FUNCTION_BLOCK GearTask IMPLEMENTS I_Task, I_Object, I_Abortable, I_Cyclic
VAR
	mcGearIn : MC_GearIn;
	mcGearOut : MC_GearOut;
	_AxisMaster : REFERENCE TO Tc2_MC2.AXIS_REF;
	_Axis : REFERENCE TO Tc2_MC2.AXIS_REF;
END_VAR

METHOD Abort : Base_Library.HRESULT
mcGearIn.Execute := FALSE;
mcGearOut.Execute := FALSE;
END_METHOD

PROPERTY PUBLIC Acceleration : mc_lreal
GET
Acceleration := mcGearIn.Acceleration;
END_GET
SET
mcGearIn.Acceleration := Acceleration;
END_SET
END_PROPERTY

PROPERTY Busy : BOOL
GET
Busy := mcGearIn.Busy OR mcGearOut.Busy;
END_GET
END_PROPERTY

METHOD Cycle : Base_Library.HRESULT
mcGearIn(Master := _AxisMaster, Slave := _Axis);
mcGearOut(Slave := _Axis);
END_METHOD

PROPERTY PUBLIC Deceleration : mc_lreal
GET
Deceleration := mcGearIn.Deceleration;
END_GET
SET
mcGearIn.Deceleration := Deceleration;
END_SET
END_PROPERTY

PROPERTY Done : BOOL
GET
Done := not mcGearIn.Busy OR NOT mcGearOut.Busy;
END_GET
END_PROPERTY

PROPERTY Error : BOOL
GET
Error := mcGearIn.Error OR mcGearOut.Error;
END_GET
END_PROPERTY

METHOD GearIn : BOOL
VAR_INPUT
END_VAR
IF _Axis.Status.NotMoving AND NOT _Axis.Status.Coupled THEN
	mcGearIn.Execute := TRUE;
END_IF
END_METHOD

METHOD GearOut : BOOL
VAR_INPUT
END_VAR
IF _Axis.Status.NotMoving AND _Axis.Status.Coupled THEN
	mcGearOut.Execute := TRUE;
END_IF
END_METHOD

PROPERTY InGear : BOOL
GET
END_GET
END_PROPERTY

PROPERTY PUBLIC Jerk : mc_lreal
GET
Jerk := mcGearIn.Jerk;
END_GET
SET
mcGearIn.Jerk := Jerk;
END_SET
END_PROPERTY

METHOD RegisterWithParent
VAR_INPUT
	Runner	: Base_Library.I_HostObjects;
END_VAR
Runner.RegisterAbortable(THIS^);
Runner.RegisterCyclic(THIS^);
Runner.RegisterTask(This^);
END_METHOD

END_FUNCTION_BLOCK

(* stored: Version 1.1.0.1
   POU GearTask: Id {c68427ee-fbb2-4955-87f7-236eb5ca7453}, SpecialFunc None
   Method Abort: Id {b070cc04-b789-4192-a434-c23424a575ce}
   Property Acceleration: Id {f01bc33a-2696-4e8f-90b9-30cdb8f4dd2d}
   Get Get: Id {b978d70b-e2e1-4621-bbee-98b107797754}
   Set Set: Id {bf531977-c15d-49ee-be06-c4bf1afca554}
   Property Busy: Id {ebe05db7-1dd0-4727-938c-463df03890a3}
   Get Get: Id {c269a663-4580-4d6d-be8e-3ee03a475cea}
   Method Cycle: Id {f8090c6e-65b8-4fad-b206-c4a3dca766fd}
   Property Deceleration: Id {92ba61af-a15e-46bf-86f4-eb6ef3fa3283}
   Get Get: Id {45a7a481-b87c-432c-a695-4c0b2d6b9967}
   Set Set: Id {1fdb4b60-2615-4d67-b857-06b44d7e0ea7}
   Property Done: Id {c8b5b359-573b-4583-94ce-5502687bec74}
   Get Get: Id {b17160ab-4958-4a0a-b824-243078353120}
   Property Error: Id {17bc1a67-dcb6-4a2a-987a-a0a1c3b242d6}
   Get Get: Id {5afed4c0-6112-40ef-95fe-e23898a97ab5}
   Method GearIn: Id {a71fc049-0a78-4bbd-8c6d-e1cd8c076d5d}
   Method GearOut: Id {7cc81acd-0a8f-4d8a-a325-58c9914d04f1}
   Property InGear: Id {7b9c5c0a-d5e8-485c-a913-d9dcff95acaf}
   Get Get: Id {90c2ce14-3a80-48f2-ac71-a190f78ea8d7}
   Property Jerk: Id {3001f9ac-1396-4b6a-8b5d-39fab90248cf}
   Get Get: Id {5e91fa52-0fff-43a5-91c7-7cdc52f5efad}
   Set Set: Id {b62bf38e-8455-4580-a928-54ae97acf0ef}
   Method RegisterWithParent: Id {3aa8e96a-b079-418b-b42d-30714fde13ef} *)
